// Mitsubishi GX Works2 project: PLC_GROUP12   PLC: FX3G

// global labels: Global1
VAR_GLOBAL
  Start_Work_Day AT X010 : BOOL;
  Oranges_Input AT D1100 : REAL;
  Tangerins_Input AT D1102 : REAL;
  Pomels_Input AT D1104 : REAL;
  Oranges_Stock AT D1106 : REAL;
  Tangerins_Stock AT D1108 : REAL;
  Pomels_Stock AT D1110 : REAL;
  Assist0 AT M0 : BOOL;
  Assist3 AT M3 : BOOL;
  Assist4 AT M4 : BOOL;
  Emergancy_Botton AT X007 : BOOL;
  Work_Day_Lamp AT Y010 : BOOL;
  Start_Wash AT X002 : BOOL;
  Washing_Container_Oranges AT D1114 : REAL;
  Washing_Container_Tangerins AT D1116 : REAL;
  Assist5 AT M8 : BOOL;
  Washing_Container_Pomels AT D1118 : REAL;
  Washing_Lamp_Timer AT TC1 : BOOL;
  Washing_Lamp_Timer_done AT TS1 : BOOL;
  Washing_Lamp AT Y005 : BOOL;
  Collecting_Lamp AT Y001 : BOOL;
  Start_Collecting AT X001 : BOOL;
  Squeeze_Container AT D1120 : REAL;
  Press_On_X11_Counter AT CC0 : BOOL;
END_VAR
VAR_GLOBAL CONSTANT
  Num_Of_Presses_Needed : INT := 2;
END_VAR
VAR_GLOBAL
  Num_Of_Presses_Done AT CS0 : BOOL;
  Squeezing_Timer AT TC2 : BOOL;
  Sqeezing_Timer_Ended AT TS2 : BOOL;
  Assist9 AT M12 : BOOL;
END_VAR
VAR_GLOBAL CONSTANT
  Const_Blink : INT := 5;
END_VAR
VAR_GLOBAL
  Blink_Timer1 AT TC3 : BOOL;
  Blink_Timer1_Ended AT TS3 : BOOL;
  Blink_Y2 AT Y002 : BOOL;
  Blink_Timer2 AT TC4 : BOOL;
  Blink_Timer2_Ended AT TS4 : BOOL;
  Blink_Y3 AT Y003 : BOOL;
  Juice_Container AT D1122 : REAL;
  Start_Quality_Test AT X003 : BOOL;
  Quality_Test_Counter AT CC1 : BOOL;
END_VAR
VAR_GLOBAL CONSTANT
  Num_Of_bad_Tests : INT := 2;
END_VAR
VAR_GLOBAL
  Test_Done AT M13 : BOOL;
END_VAR
VAR_GLOBAL CONSTANT
  Test_Min_Val : REAL := 1;
  Test_Max_Val : REAL := 5;
END_VAR
VAR_GLOBAL
  Quality_Test_OK AT M14 : BOOL;
  Quality_Test_NOT_OK AT M15 : BOOL;
  Succsess_Lamp_Timer AT TC5 : BOOL;
  Succsess_Lamp_Timer_Ended AT TS5 : BOOL;
END_VAR
VAR_GLOBAL CONSTANT
  Success_Lamp_Time : INT := 50;
END_VAR
VAR_GLOBAL
  Test_OK_Lamp AT Y004 : BOOL;
  Juice_Storage AT D1126 : REAL;
END_VAR
VAR_GLOBAL CONSTANT
  Zero_Const : REAL;
END_VAR
VAR_GLOBAL
  Quality_Test_Counter_ReachedMAX AT CS1 : BOOL;
  End_Day AT M16 : BOOL;
END_VAR
VAR_GLOBAL CONSTANT
  Const_Min_To_Supply : REAL := 150;
END_VAR
VAR_GLOBAL
  Available_To_Supply AT Y006 : BOOL;
END_VAR
VAR_GLOBAL CONSTANT
  Const_Handred : REAL := 100;
END_VAR
VAR_GLOBAL
  Supply AT X004 : BOOL;
  Supplier_Demand AT D1128 : REAL;
  Amount_To_Supply AT D1130 : REAL;
  Supplied AT M17 : BOOL;
  Juice_Quality_Test_Result_Float AT D1132 : REAL;
END_VAR
VAR_GLOBAL CONSTANT
  Const_4 : REAL := 4;
END_VAR
VAR_GLOBAL
  Analog_Input_2 AT D8281 : INT;
  Max_Tangerins_Pomels_available AT D1124 : REAL;
END_VAR
VAR_GLOBAL CONSTANT
  Const_Two : REAL := 2;
END_VAR
VAR_GLOBAL
  Max_Oranges_Needed AT D1134 : REAL;
  Oranges_Amount_Before_Limitation AT D1136 : REAL;
  Oranges_Amount_To_Production AT D1138 : REAL;
  Pomels_Amount_To_Production AT D1140 : REAL;
  Tangerins_Amount_To_Production AT D1142 : REAL;
  Assist30 AT M30 : BOOL;
  In_Washing_Stage AT M31 : BOOL;
  End_Washing_Stage AT M33 : BOOL;
  End_Collection_Stage AT M34 : BOOL;
  In_Squeezing_Stage AT M35 : BOOL;
  End_Squeezing_Stage AT M36 : BOOL;
  End_Quality_Stage_Test_OK AT M37 : BOOL;
  End_Quality_Stage_Test_NOT_OK AT M38 : BOOL;
  End_Of_Iteration AT M40 : BOOL;
  Stock_Check_OK AT M50 : BOOL;
  Stock_Check_NOT_OK AT M51 : BOOL;
  End_Quality_Stage AT M43 : BOOL;
  Control_Blink_End_Day AT M22 : BOOL;
  Blinking_End_Day_Timer AT TC6 : BOOL;
  End_Day_Timer_Ended AT TS6 : BOOL;
  Blink_Asist1 AT M18 : BOOL;
  Blink_Asist2 AT M19 : BOOL;
  Analog_Output AT D8282 : INT;
END_VAR
VAR_GLOBAL CONSTANT
  Const_400 : REAL := 400;
END_VAR
VAR_GLOBAL
  Count_First_Iteration AT CC2 : BOOL;
END_VAR
VAR_GLOBAL CONSTANT
  One_Iteration : INT := 1;
END_VAR
VAR_GLOBAL
  Count_First_Iteration_Ended AT CS2 : BOOL;
  Start_Squeezing AT X011 : BOOL;
END_VAR
VAR_GLOBAL CONSTANT
  Const_3 : INT := 30;
END_VAR

// task Task_01 (event TRUE, interval 0, priority 31): POU_01

PROGRAM POU_01
(* structured ladder/FBD written out as ST: instructions are called as NAME(EN, inputs, outputs); _pN, _eN, _tN stand for wires *)
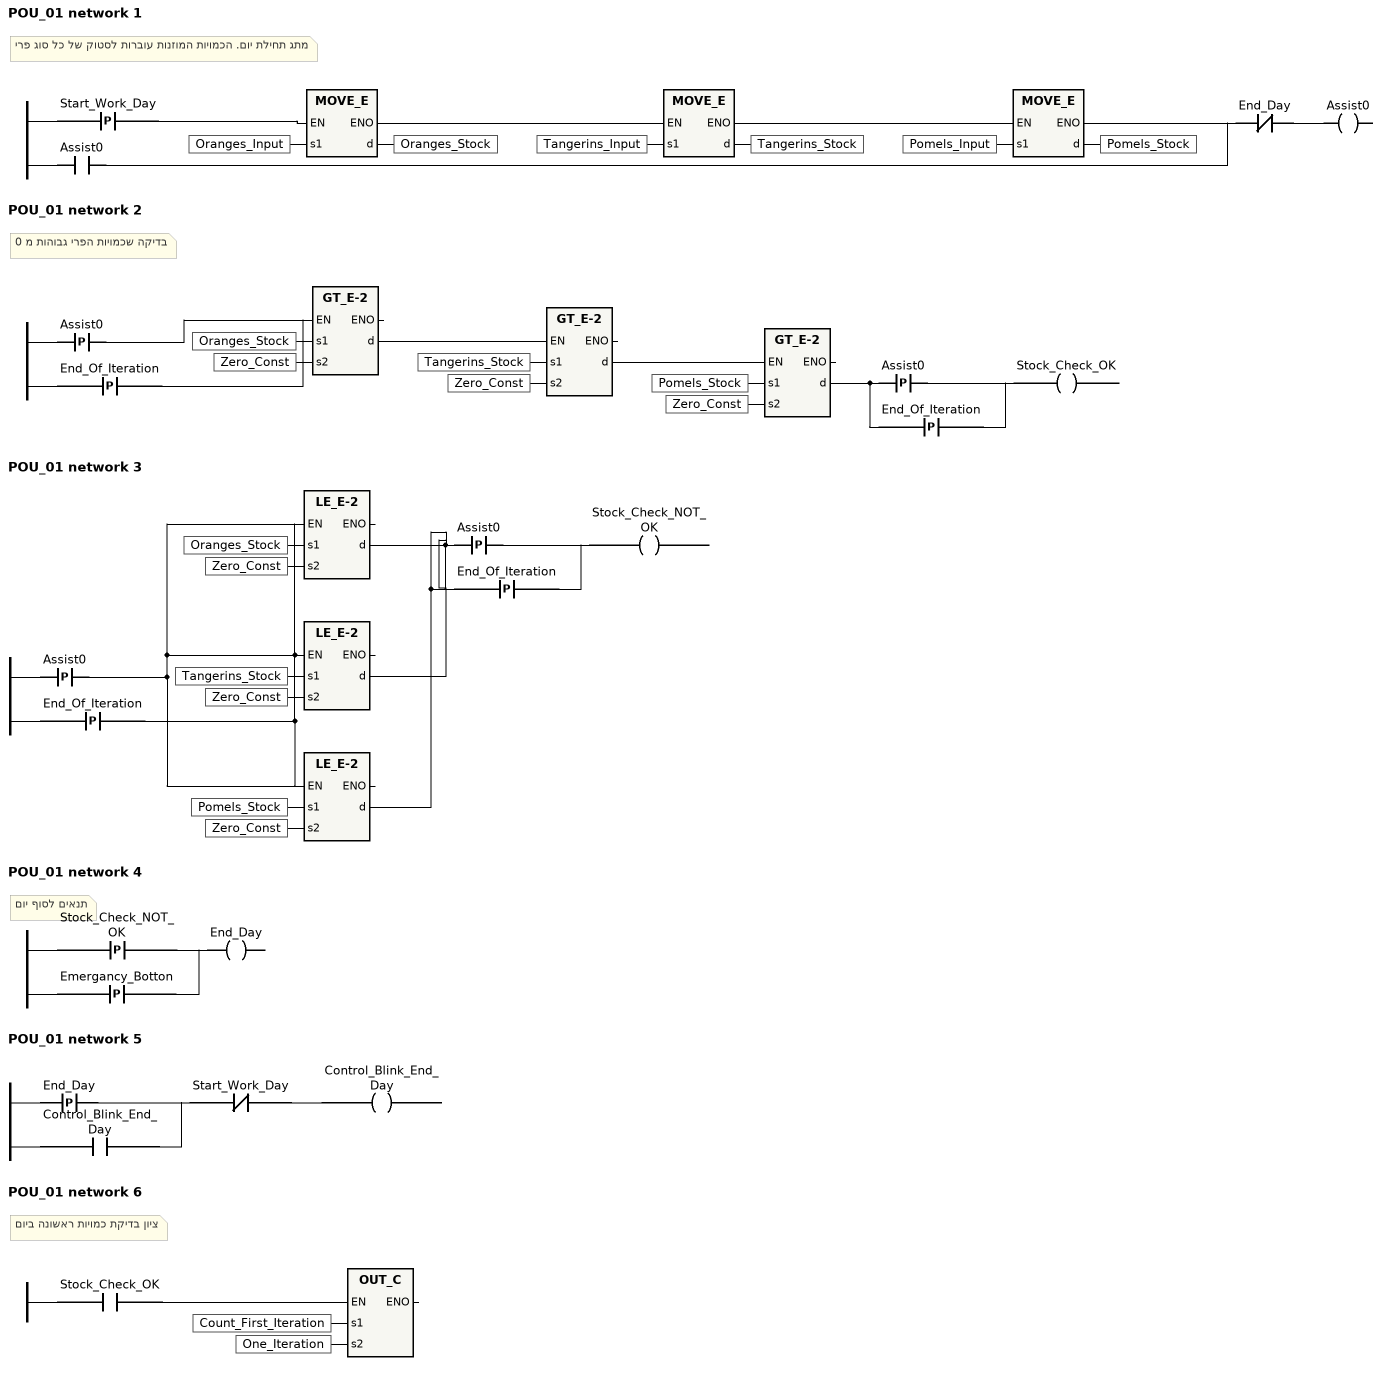
(* network 1 *)
(* מתג תחילת יום. הכמויות המוזנות עוברות לסטוק של כל סוג פרי *)
_e1 := MOVE_E(LDP(TRUE, Start_Work_Day), Oranges_Input, Oranges_Stock);
_e2 := MOVE_E(_e1, Tangerins_Input, Tangerins_Stock);
_e3 := MOVE_E(_e2, Pomels_Input, Pomels_Stock);
Assist0 := (_e3 OR Assist0) AND NOT End_Day;
(* network 2 *)
(* בדיקה שכמויות הפרי גבוהות מ 0 *)
GT_E(LDP(TRUE, Assist0) OR LDP(TRUE, End_Of_Iteration), Oranges_Stock, Zero_Const, _t1);
GT_E(_t1, Tangerins_Stock, Zero_Const, _t2);
GT_E(_t2, Pomels_Stock, Zero_Const, _t3);
Stock_Check_OK := (_t3 AND LDP(TRUE, Assist0)) OR (_t3 AND LDP(TRUE, End_Of_Iteration));
(* network 3 *)
_p1 := LDP(TRUE, Assist0) OR LDP(TRUE, End_Of_Iteration);
LE_E(_p1, Oranges_Stock, Zero_Const, _t2);
LE_E(_p1, Tangerins_Stock, Zero_Const, _t3);
LE_E(_p1, Pomels_Stock, Zero_Const, _t4);
_p5 := _t2 OR _t3 OR _t4;
Stock_Check_NOT_OK := (_p5 AND LDP(TRUE, Assist0)) OR (_p5 AND LDP(TRUE, End_Of_Iteration));
(* network 4 *)
(* תנאים לסוף יום *)
End_Day := LDP(TRUE, Stock_Check_NOT_OK) OR LDP(TRUE, Emergancy_Botton);
(* network 5 *)
Control_Blink_End_Day := (LDP(TRUE, End_Day) OR Control_Blink_End_Day) AND NOT Start_Work_Day;
(* network 6 *)
(* ציון בדיקת כמויות ראשונה ביום *)
OUT_C(Stock_Check_OK, Count_First_Iteration, One_Iteration);
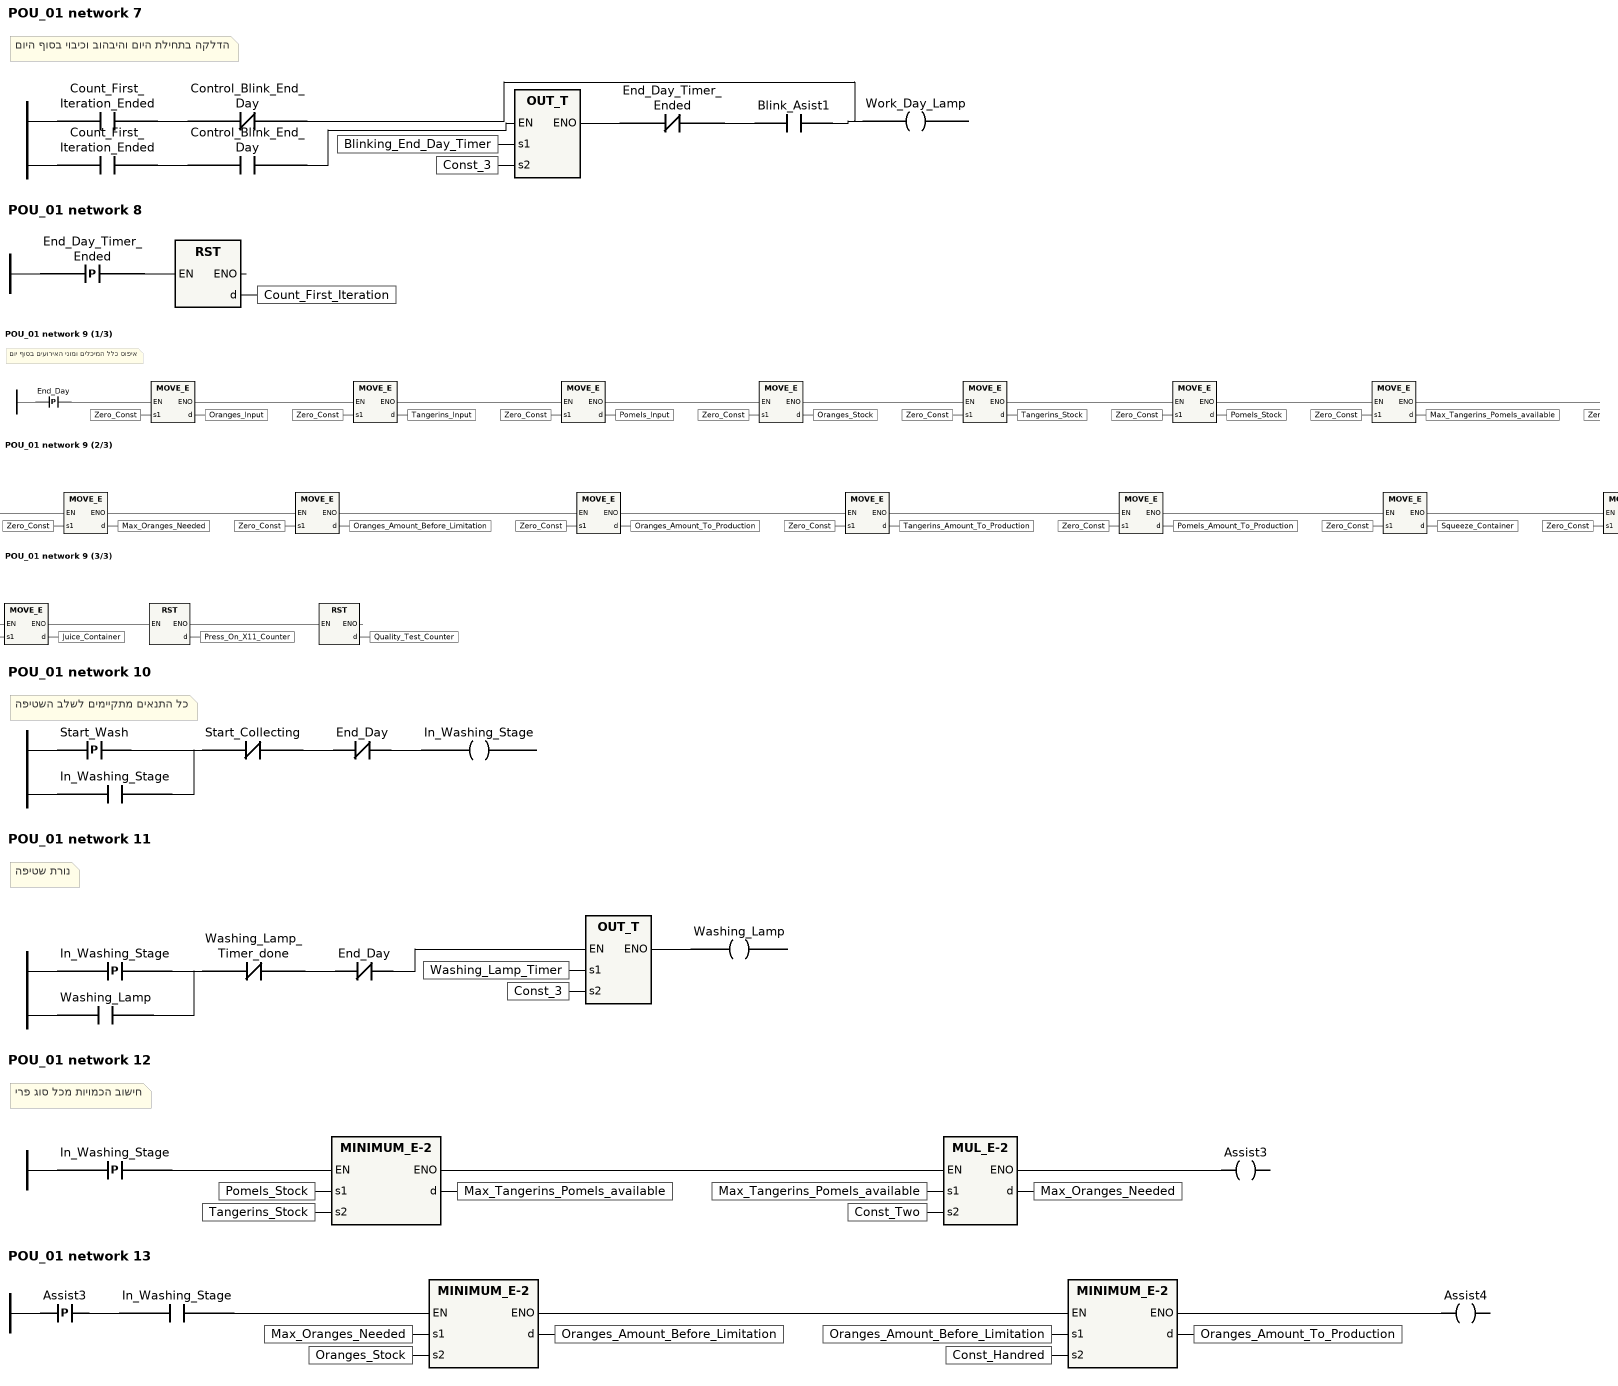
(* network 7 *)
(* הדלקה בתחילת היום והיבהוב וכיבוי בסוף היום *)
_e1 := OUT_T(Count_First_Iteration_Ended AND Control_Blink_End_Day, Blinking_End_Day_Timer, Const_3);
Work_Day_Lamp := (Count_First_Iteration_Ended AND NOT Control_Blink_End_Day) OR (_e1 AND NOT End_Day_Timer_Ended AND Blink_Asist1);
(* network 8 *)
RST(LDP(TRUE, End_Day_Timer_Ended), Count_First_Iteration);
(* network 9 *)
(* איפוס כלל המיכלים ומוני האירועים בסוף יום *)
_e1 := MOVE_E(LDP(TRUE, End_Day), Zero_Const, Oranges_Input);
_e2 := MOVE_E(_e1, Zero_Const, Tangerins_Input);
_e3 := MOVE_E(_e2, Zero_Const, Pomels_Input);
_e4 := MOVE_E(_e3, Zero_Const, Oranges_Stock);
_e5 := MOVE_E(_e4, Zero_Const, Tangerins_Stock);
_e6 := MOVE_E(_e5, Zero_Const, Pomels_Stock);
_e7 := MOVE_E(_e6, Zero_Const, Max_Tangerins_Pomels_available);
_e8 := MOVE_E(_e7, Zero_Const, Max_Oranges_Needed);
_e9 := MOVE_E(_e8, Zero_Const, Oranges_Amount_Before_Limitation);
_e10 := MOVE_E(_e9, Zero_Const, Oranges_Amount_To_Production);
_e11 := MOVE_E(_e10, Zero_Const, Tangerins_Amount_To_Production);
_e12 := MOVE_E(_e11, Zero_Const, Pomels_Amount_To_Production);
_e13 := MOVE_E(_e12, Zero_Const, Squeeze_Container);
_e14 := MOVE_E(_e13, Zero_Const, Juice_Container);
_e15 := RST(_e14, Press_On_X11_Counter);
RST(_e15, Quality_Test_Counter);
(* network 10 *)
(* כל התנאים מתקיימים לשלב השטיפה *)
In_Washing_Stage := ((LDP(TRUE, Start_Wash) OR In_Washing_Stage) AND NOT Start_Collecting) AND NOT End_Day;
(* network 11 *)
(* נורת שטיפה *)
_e1 := OUT_T(((LDP(TRUE, In_Washing_Stage) OR Washing_Lamp) AND NOT Washing_Lamp_Timer_done) AND NOT End_Day, Washing_Lamp_Timer, Const_3);
Washing_Lamp := _e1;
(* network 12 *)
(* חישוב הכמויות מכל סוג פרי *)
_e1 := MINIMUM_E(LDP(TRUE, In_Washing_Stage), Pomels_Stock, Tangerins_Stock, Max_Tangerins_Pomels_available);
_e2 := MUL_E(_e1, Max_Tangerins_Pomels_available, Const_Two, Max_Oranges_Needed);
Assist3 := _e2;
(* network 13 *)
_e1 := MINIMUM_E(LDP(TRUE, Assist3) AND In_Washing_Stage, Max_Oranges_Needed, Oranges_Stock, Oranges_Amount_Before_Limitation);
_e2 := MINIMUM_E(_e1, Oranges_Amount_Before_Limitation, Const_Handred, Oranges_Amount_To_Production);
Assist4 := _e2;
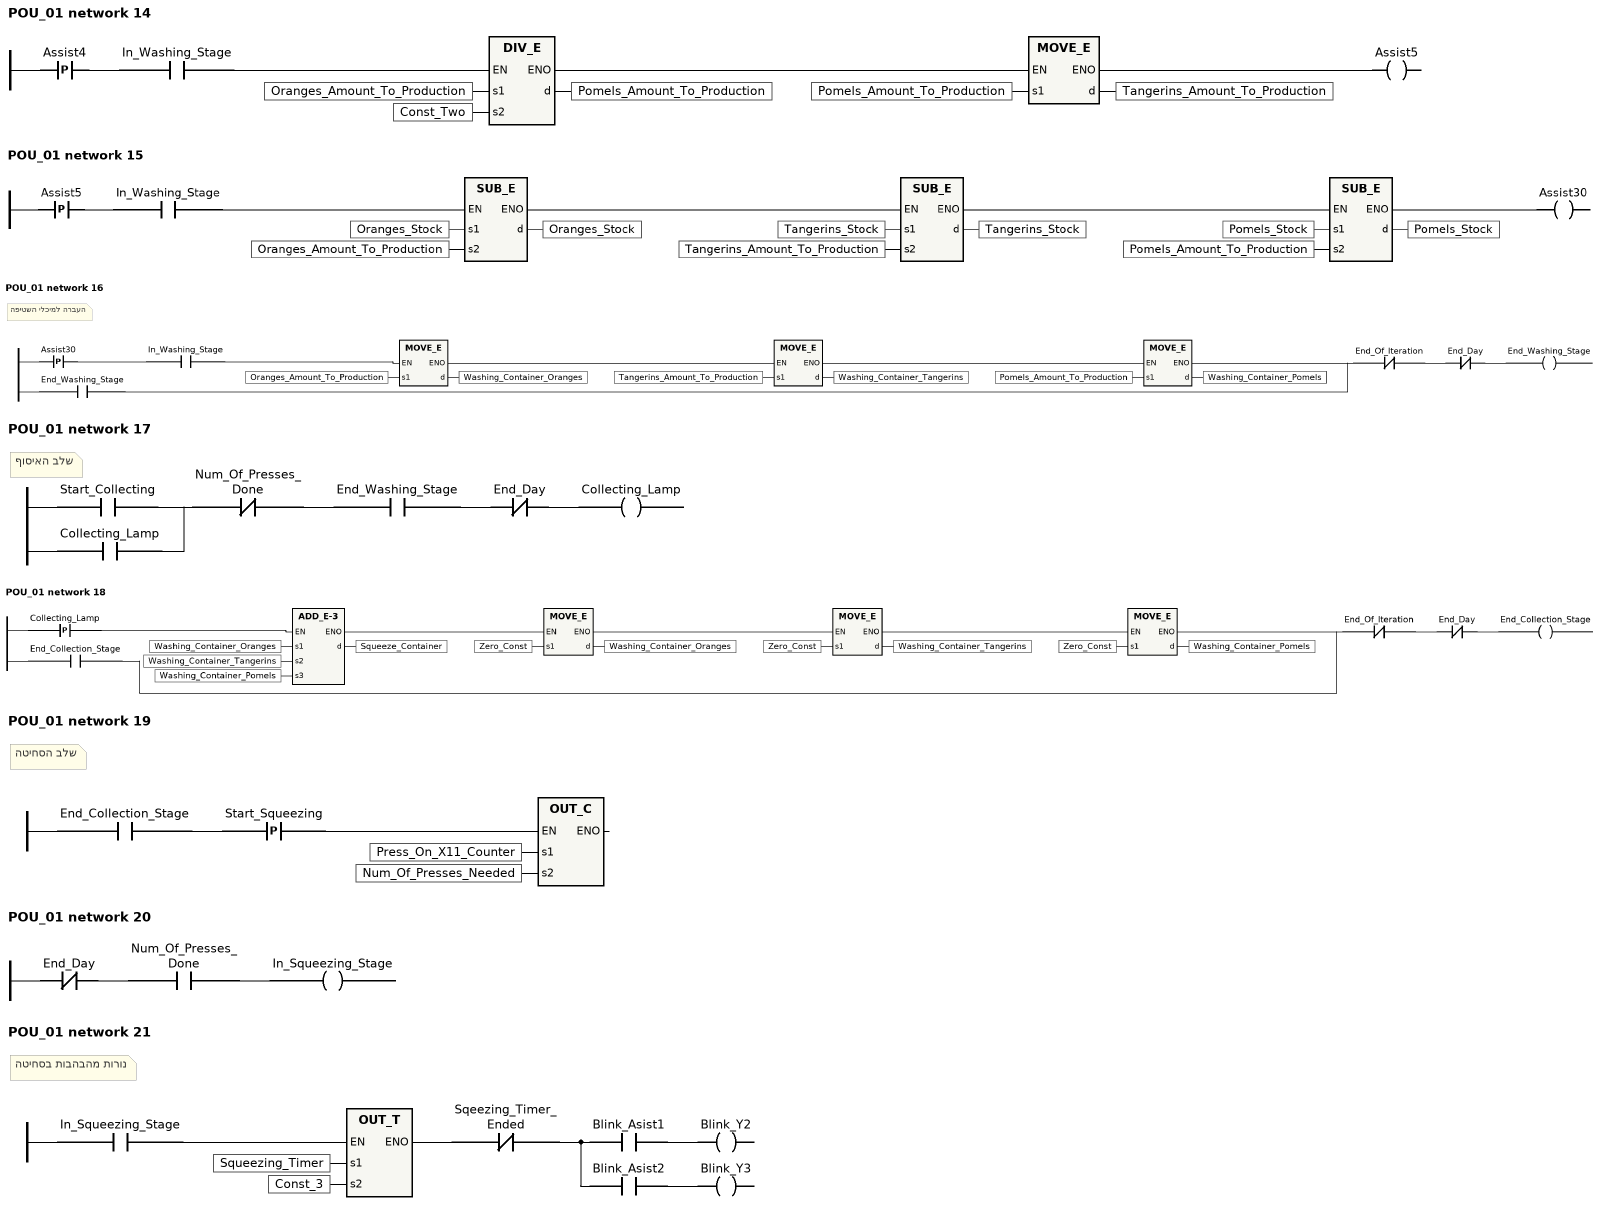
(* network 14 *)
_e1 := DIV_E(LDP(TRUE, Assist4) AND In_Washing_Stage, Oranges_Amount_To_Production, Const_Two, Pomels_Amount_To_Production);
_e2 := MOVE_E(_e1, Pomels_Amount_To_Production, Tangerins_Amount_To_Production);
Assist5 := _e2;
(* network 15 *)
_e1 := SUB_E(LDP(TRUE, Assist5) AND In_Washing_Stage, Oranges_Stock, Oranges_Amount_To_Production, Oranges_Stock);
_e2 := SUB_E(_e1, Tangerins_Stock, Tangerins_Amount_To_Production, Tangerins_Stock);
_e3 := SUB_E(_e2, Pomels_Stock, Pomels_Amount_To_Production, Pomels_Stock);
Assist30 := _e3;
(* network 16 *)
(* העברה למיכלי השטיפה *)
_e1 := MOVE_E(LDP(TRUE, Assist30) AND In_Washing_Stage, Oranges_Amount_To_Production, Washing_Container_Oranges);
_e2 := MOVE_E(_e1, Tangerins_Amount_To_Production, Washing_Container_Tangerins);
_e3 := MOVE_E(_e2, Pomels_Amount_To_Production, Washing_Container_Pomels);
End_Washing_Stage := ((_e3 OR End_Washing_Stage) AND NOT End_Of_Iteration) AND NOT End_Day;
(* network 17 *)
(* שלב האיסוף *)
Collecting_Lamp := (((Start_Collecting OR Collecting_Lamp) AND NOT Num_Of_Presses_Done) AND End_Washing_Stage) AND NOT End_Day;
(* network 18 *)
_e1 := ADD_E(LDP(TRUE, Collecting_Lamp), Washing_Container_Oranges, Washing_Container_Tangerins, Washing_Container_Pomels, Squeeze_Container);
_e2 := MOVE_E(_e1, Zero_Const, Washing_Container_Oranges);
_e3 := MOVE_E(_e2, Zero_Const, Washing_Container_Tangerins);
_e4 := MOVE_E(_e3, Zero_Const, Washing_Container_Pomels);
End_Collection_Stage := ((_e4 OR End_Collection_Stage) AND NOT End_Of_Iteration) AND NOT End_Day;
(* network 19 *)
(* שלב הסחיטה *)
OUT_C(End_Collection_Stage AND LDP(TRUE, Start_Squeezing), Press_On_X11_Counter, Num_Of_Presses_Needed);
(* network 20 *)
In_Squeezing_Stage := NOT End_Day AND Num_Of_Presses_Done;
(* network 21 *)
(* נורות מהבהבות בסחיטה *)
_e1 := OUT_T(In_Squeezing_Stage, Squeezing_Timer, Const_3);
_p2 := _e1 AND NOT Sqeezing_Timer_Ended;
Blink_Y2 := _p2 AND Blink_Asist1;
Blink_Y3 := _p2 AND Blink_Asist2;
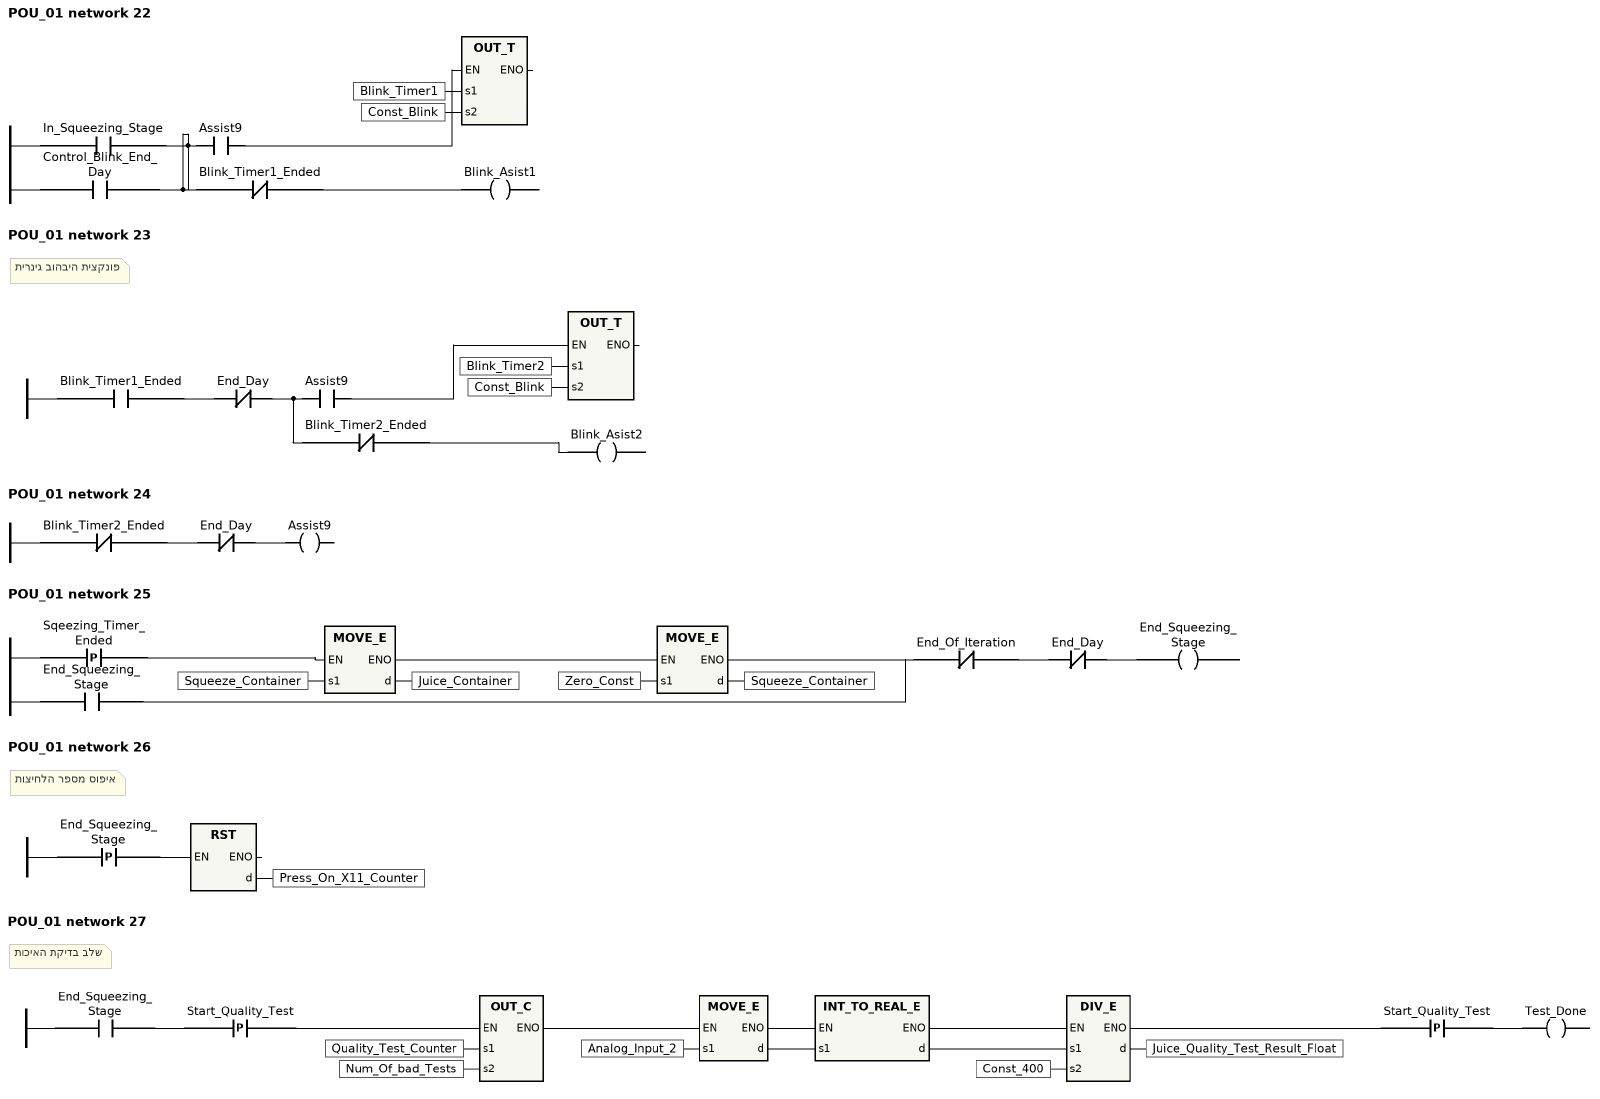
(* network 22 *)
_p1 := In_Squeezing_Stage OR Control_Blink_End_Day;
OUT_T(_p1 AND Assist9, Blink_Timer1, Const_Blink);
Blink_Asist1 := _p1 AND NOT Blink_Timer1_Ended;
(* network 23 *)
(* פונקצית היבהוב גינרית *)
_p1 := Blink_Timer1_Ended AND NOT End_Day;
OUT_T(_p1 AND Assist9, Blink_Timer2, Const_Blink);
Blink_Asist2 := _p1 AND NOT Blink_Timer2_Ended;
(* network 24 *)
Assist9 := NOT Blink_Timer2_Ended AND NOT End_Day;
(* network 25 *)
_e1 := MOVE_E(LDP(TRUE, Sqeezing_Timer_Ended), Squeeze_Container, Juice_Container);
_e2 := MOVE_E(_e1, Zero_Const, Squeeze_Container);
End_Squeezing_Stage := ((_e2 OR End_Squeezing_Stage) AND NOT End_Of_Iteration) AND NOT End_Day;
(* network 26 *)
(* איפוס מספר הלחיצות *)
RST(LDP(TRUE, End_Squeezing_Stage), Press_On_X11_Counter);
(* network 27 *)
(* שלב בדיקת האיכות *)
_e1 := OUT_C(End_Squeezing_Stage AND LDP(TRUE, Start_Quality_Test), Quality_Test_Counter, Num_Of_bad_Tests);
_e3 := MOVE_E(_e1, Analog_Input_2, _t2);
_e5 := INT_TO_REAL_E(_e3, _t2, _t4);
_e6 := DIV_E(_e5, _t4, Const_400, Juice_Quality_Test_Result_Float);
Test_Done := _e6 AND LDP(TRUE, Start_Quality_Test);
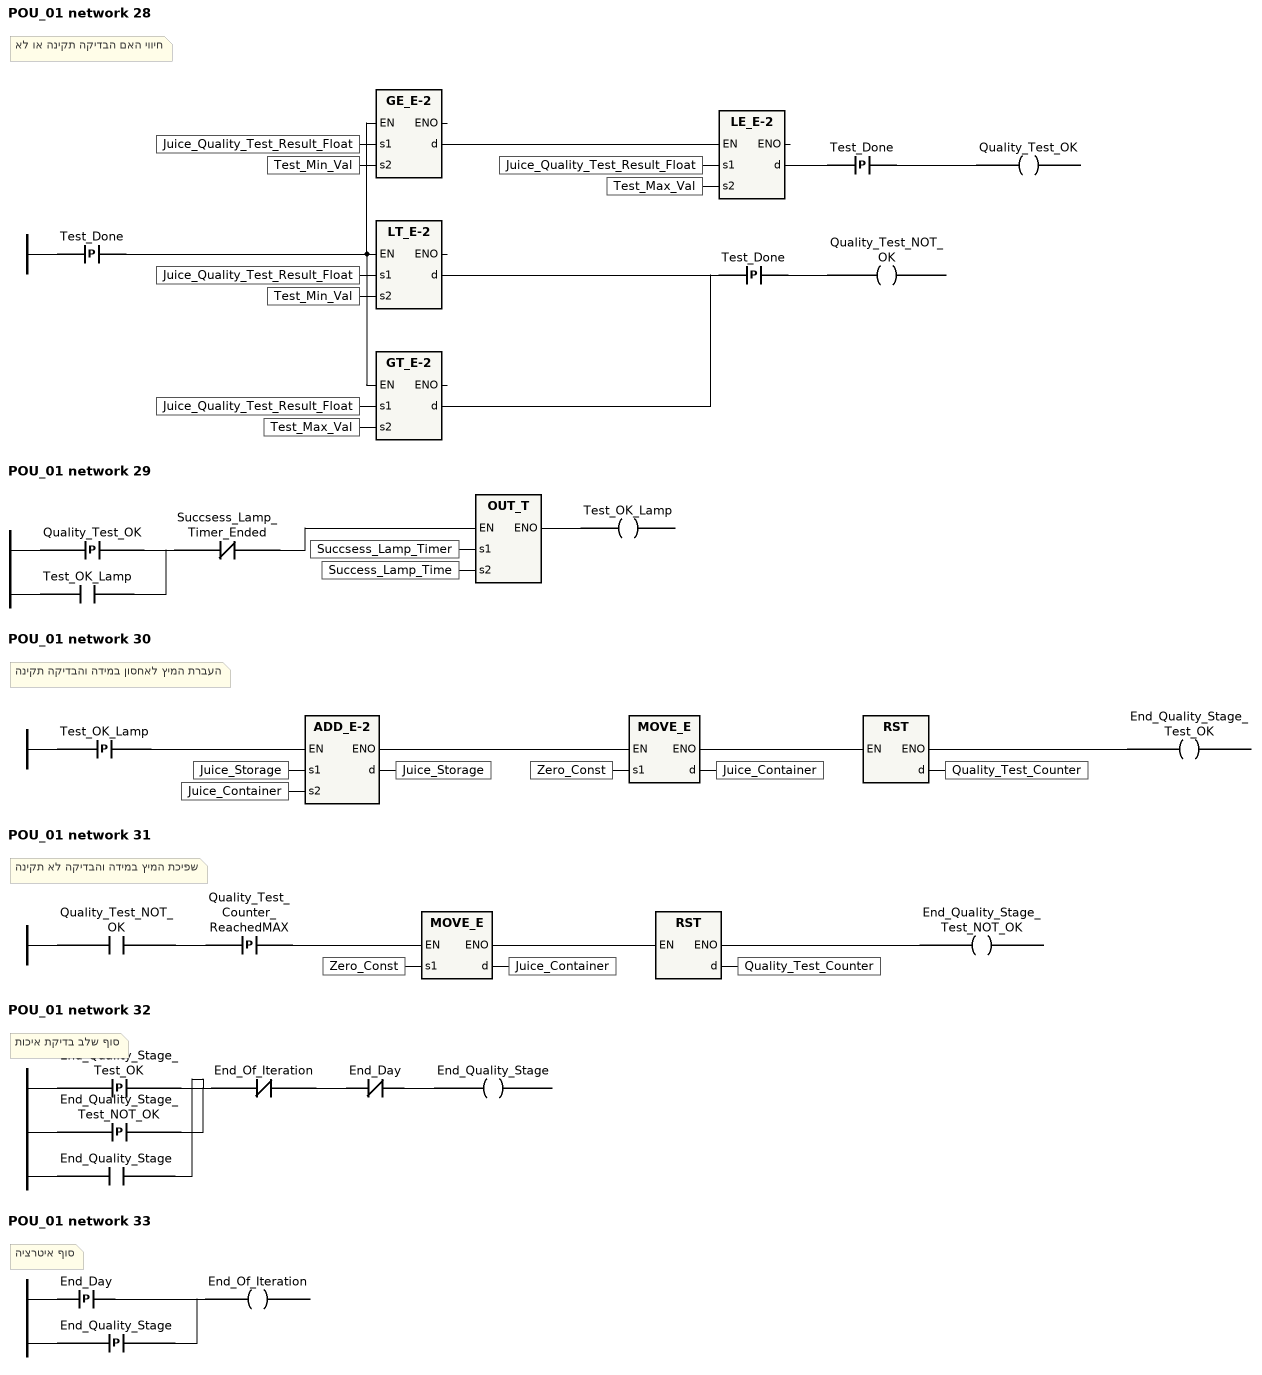
(* network 28 *)
(* חיווי האם הבדיקה תקינה או לא *)
_p1 := LDP(TRUE, Test_Done);
GE_E(_p1, Juice_Quality_Test_Result_Float, Test_Min_Val, _t2);
LE_E(_t2, Juice_Quality_Test_Result_Float, Test_Max_Val, _t3);
Quality_Test_OK := _t3 AND LDP(TRUE, Test_Done);
LT_E(_p1, Juice_Quality_Test_Result_Float, Test_Min_Val, _t4);
GT_E(_p1, Juice_Quality_Test_Result_Float, Test_Max_Val, _t5);
Quality_Test_NOT_OK := (_t4 OR _t5) AND LDP(TRUE, Test_Done);
(* network 29 *)
_e1 := OUT_T((LDP(TRUE, Quality_Test_OK) OR Test_OK_Lamp) AND NOT Succsess_Lamp_Timer_Ended, Succsess_Lamp_Timer, Success_Lamp_Time);
Test_OK_Lamp := _e1;
(* network 30 *)
(* העברת המיץ לאחסון במידה והבדיקה תקינה *)
_e1 := ADD_E(LDP(TRUE, Test_OK_Lamp), Juice_Storage, Juice_Container, Juice_Storage);
_e2 := MOVE_E(_e1, Zero_Const, Juice_Container);
_e3 := RST(_e2, Quality_Test_Counter);
End_Quality_Stage_Test_OK := _e3;
(* network 31 *)
(* שפיכת המיץ במידה והבדיקה לא תקינה *)
_e1 := MOVE_E(Quality_Test_NOT_OK AND LDP(TRUE, Quality_Test_Counter_ReachedMAX), Zero_Const, Juice_Container);
_e2 := RST(_e1, Quality_Test_Counter);
End_Quality_Stage_Test_NOT_OK := _e2;
(* network 32 *)
(* סוף שלב בדיקת איכות *)
End_Quality_Stage := ((LDP(TRUE, End_Quality_Stage_Test_OK) OR LDP(TRUE, End_Quality_Stage_Test_NOT_OK) OR End_Quality_Stage) AND NOT End_Of_Iteration) AND NOT End_Day;
(* network 33 *)
(* סוף איטרציה *)
End_Of_Iteration := LDP(TRUE, End_Day) OR LDP(TRUE, End_Quality_Stage);
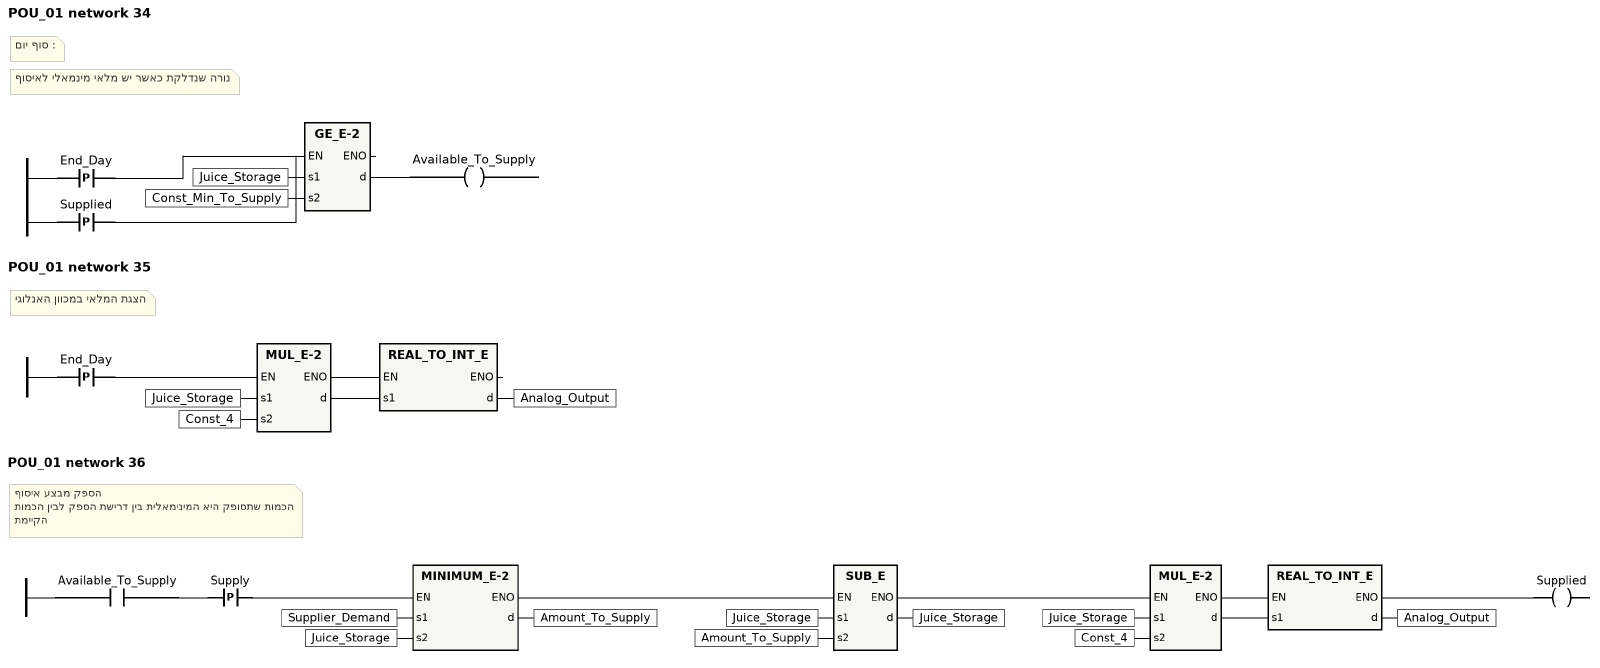
(* network 34 *)
(* : סוף יום *)
(* נורה שנדלקת כאשר יש מלאי מינמאלי לאיסוף *)
GE_E(LDP(TRUE, End_Day) OR LDP(TRUE, Supplied), Juice_Storage, Const_Min_To_Supply, _t1);
Available_To_Supply := _t1;
(* network 35 *)
(* הצגת המלאי במכוון האנלוגי *)
_e2 := MUL_E(LDP(TRUE, End_Day), Juice_Storage, Const_4, _t1);
REAL_TO_INT_E(_e2, _t1, Analog_Output);
(* network 36 *)
(* הספק מבצע איסוף / הכמות שתסופק היא המינימאלית בין דרישת הספק לבין הכמות הקיימת *)
_e1 := MINIMUM_E(Available_To_Supply AND LDP(TRUE, Supply), Supplier_Demand, Juice_Storage, Amount_To_Supply);
_e2 := SUB_E(_e1, Juice_Storage, Amount_To_Supply, Juice_Storage);
_e4 := MUL_E(_e2, Juice_Storage, Const_4, _t3);
_e5 := REAL_TO_INT_E(_e4, _t3, Analog_Output);
Supplied := _e5;
END_PROGRAM
